(*
An identifier that uses reflection to generate a unique symbol path.
It simplifies the path by removing project, PLC, and tag segments.
Example:
- Reflection: proj.plc.MAIN.functionBlock[*]._tag
- Path: MAIN.functionBlock.5
*)
{attribute 'reflection'}
FUNCTION_BLOCK TagBase IMPLEMENTS I_Tag
VAR
	{attribute 'instance-path'} 
    {attribute 'noinit'} 
	_sId			: Str;
	_nOptionPos		: USINT;
	_nOptionLen		: USINT;
END_VAR

{attribute 'hide'}
METHOD FB_init : BOOL
VAR_INPUT
	bInitRetains : BOOL; // if TRUE, the retain variables are initialized (warm start / cold start)
	bInCopyCode : BOOL;  // if TRUE, the instance afterwards gets moved into the copy code (online change)
END_VAR
VAR
	i				: INT;
	_sChar			: Ch;
END_VAR
// Delete this name
FOR i := Tc2_Standard.LEN(_sId) TO 1 BY -1 DO
	IF Tc2_Standard.MID(_sId, 1, i) = '.' THEN
		_sId := Tc2_Standard.LEFT(_sId, i - 1);
		EXIT;
	END_IF
END_FOR

// Delete project name
FOR i := 1 TO Tc2_Standard.LEN(_sId) DO
	IF Tc2_Standard.MID(_sId, 1, i) = '.' THEN
		_sId := Tc2_Standard.DELETE(_sId, i, 1);
		EXIT;
	END_IF
END_FOR

// Delete plc name
FOR i := 1 TO Tc2_Standard.LEN(_sId) DO
	IF Tc2_Standard.MID(_sId, 1, i) = '.' THEN
		_sId := Tc2_Standard.DELETE(_sId, i, 1);
		EXIT;
	END_IF
END_FOR

// Replace '[' with '.' and remove ']' 
FOR i := 1 TO Tc2_Standard.LEN(_sId) DO
	_sChar := Tc2_Standard.MID(_sId, 1, i);
	IF _sChar = '[' THEN
		_sId := Tc2_Standard.REPLACE(_sId, '.', 1, i);
	ELSIF _sChar = ']' THEN
		_sId := Tc2_Standard.DELETE(_sId, 1, i);
	END_IF
END_FOR

_sId := Tc2_Utilities.F_ToLCase(_sID);
END_METHOD

// Read address path without Option segment.
PROPERTY Id : Str
GET
IF _nOptionPos <> 0 THEN
	Id := Tc2_Standard.DELETE(_sId, _nOptionLen + 1, _nOptionPos); 
ELSE
	Id := _sId;
END_IF
END_GET
END_PROPERTY

// Modify or read the optional segment.
PROPERTY Option : Str
GET
VAR
	i				: INT;
END_VAR
IF _nOptionPos <> 0 THEN
	Option := Tc2_Standard.DELETE(_sId, _nOptionPos, 1); 
ELSE
	Option := '';
END_IF
END_GET
SET
IF Option <> '' THEN
    _nOptionLen := INT_TO_USINT(Tc2_Standard.LEN(Option));    
    IF _nOptionPos <> 0 THEN
        _sId := Tc2_Standard.LEFT(_sId, _nOptionPos);
        _sId := Tc2_Standard.CONCAT(_sId, Option);
    ELSE
        // The option does not exist, so we append it
        _nOptionPos := INT_TO_USINT(Tc2_Standard.LEN(_sId) + 1);
        _sId := Tc2_Standard.CONCAT(_sId, '.');
        _sId := Tc2_Standard.CONCAT(_sId, Option);
    END_IF
ELSIF _nOptionPos <> 0 THEN
    _sId := Tc2_Standard.LEFT(_sId, _nOptionPos - 1);
    _nOptionPos := 0;
END_IF
END_SET
END_PROPERTY

PROPERTY Proxy : REFERENCE TO I_Tag
SET
Proxy := THIS^;
END_SET
END_PROPERTY

// Return interface pointer to THIS^.
PROPERTY Self : I_Tag
GET
Self := THIS^;
END_GET
END_PROPERTY

END_FUNCTION_BLOCK

(* stored: Version 1.1.0.1
   POU TagBase: Id {2e4b93ca-cf29-4297-8c18-30aee9f4dbcc}, SpecialFunc None
   Method FB_init: Id {32f06f41-7774-4492-bbae-9ef87fedb467}
   Property Id: Id {b0dd2c0b-7dc9-43ce-98fa-e7469eee6720}
   Get Get: Id {ef9dbdd5-51da-4e00-9df9-abd90d96465d}
   Property Option: Id {66edb463-3b71-4c89-b966-006f5d753148}
   Get Get: Id {f548895c-1f6d-4c8a-932c-8d8c4861861c}
   Set Set: Id {b7ab1309-6936-40d7-9d51-047baede1f20}
   Property Proxy: Id {f27cd52a-cc58-40ed-b243-65041daea015}
   Set Set: Id {0b0052f6-98c0-4255-8c6f-f4b582b0030b}
   Property Self: Id {e153ed58-4e18-467d-9035-8a08187af0e1}
   Get Get: Id {206a24c8-8314-4d48-9be0-59b3e98c552f} *)
